# B&R Automation Studio project TD52 (part 97)

#### EG_ScavCyclic.st
```iecst
(*******************************************************************************
EG_Scav			exhaust gas scavenging + N2 scavenging

This code is confidential and proprietary to the INNIO Company.
It may not be used in any form, or reproduced in any manner,
without the express written permission of the INNIO Company.
Copyright, INNIO Company, 2022

Customized modifications: -
------------------------

History:
-------
V06		24.03.2000	PA			erstellt
V11		04.07.2000	Pa			Stoerungsaufbereitung von p10 verschoben
V160	13.12.2001	LH			Ansteuerung Spuelventilator auch mit Gasventile offen
V170	04.02.2002	LH			Moeglichkeit Spuelung manuell zu starten
V190	10.05.2004	LH			Anpassung fuer CODINOX
 								Fehler bei manueller Spuelung ausgebessert
V212	06.06.2006	LH			angepasst an ESY-NEU
V230	12.12.2007	TW			Spuelzeit ist nun Parameter (ssTW_T_SPUEL)
	 	30.01.2008	LH			Untergrenze für Spülzeit ist 47sec
V3.20.0	04.11.2010	lettenb.	purgecycle added, task spuelung renamed to spuelung_6
		14.01.2011 				sel_EGScav_if_AuxV_ok added, release exhaust gas scavenging depending on auxiliaries voltage

V1.70.1	20.03.2003	ThJ			Erweiterung auf N2-Spuelung
V1.70.2	04.05.2004	ThJ			Erweiterung N2-Spuelung von Baureihe 6 auf alle Baureihen
V1.70.3	10.11.2004	ThJ			steps 5 + 8: M_SPUELV hinzu fuer BR234
V1.70.4	15.05.2006	ThJ			Vorbelegung Option "two N2 valves" mit FALSE.
       		              		xx_T71 --> xx_TOF71, xx_T_SPUEL --> xx_TON_SPUEL.
V1.70.5	28.07.2006	ThJ			TwoN2Valves --> global, ANF_SPLV_MAN added,
       		              		N2 gas valves output, N2 valves position faulure modified.
V1.70.6	22.11.2007	ThJ			timer for reset SP_EIN / LUE100
                        		T1_SCAV_RUN: timer 80 --> 75 sec
                        		SCAV_RUN_STOE with filter BWS_A
                        		reset SCAV_RUN at BWS_H by STOP
V1.70.7 03.12.2008	lettenb. 	sel_N2, sel_TwoN2Valves added
V3.40.0	19.12.2012  lettenb.	T1_SCAV_RUN: SCAV_RUN --> STARTER_SC, PT: 75s --> 5s
.								(ueberwachung nun nicht mehr abhaengig von vorschmierzeit/motortemp...., test: SACC, leitner christian)
V3.90.0	25.10.2012	lettenb.	xTON_AuxDemDelayed, Para.bEGScav_Active added
V3.99.0	17.04.2012	lettenb.	EG scav.with all time running fan
		14.05.2013				EG scav.activation for BR6,9 added
		23.10.2013				624: delayed auxiliaries demand with EG scavenging
		28.10.2013				changes from V3.40.1 included, saver case (open flap and fan not demanded) solved
								reset manual scavenging from engine stop button changed > scav.stop button
								N2 scavenging and exhaust gas scavenging merged
		16.01.2014	lettenb.	V3.50 exh.gas scavenging after engine stop with gas train test added
		26.02.2014				tAuxV_Eng_ok.Di added, bugfix
V4.00.0	22.05.2014	lettenb.	T1_STSPKL: scav.valve monitoring open/closed status added, bugfix
V4.00.1 14.07.2014				NoScavFlap, NoScavFan: default = FALSE for EG scav.
		06.08.2014				reset VIS2MM.bN2ScavStart/Stop buttons added
		12.09.2014				SPUEL_ST: AND NOT OUT_EX.bScavFinished added(purge cycle: lock scav.during eng.oper.with eng.dem. off/on)
V4.00.2 30.10.2014	lettenb.	SPUEL_ST: OUT_EX.bScavFinished -> M_DREHZ (purge cycle: lock scav.during eng.oper.)
V4.00.3	20.03.2015	lettenb.	ScavValve opens after bScavFanOp=TRUE, ScavFanCoOn if ScavValve=open or not closed,
								3366 during purge -> close ScavValve(safety case:PW-ER-2015-0062-001)
		14.04.2015				corr.from test EG_Scav with purgecycle and/or purge before start(panian,glantschnig)
		30.04.2015 				OUT_EX.tScavFanCoOn.Do:	IN_EX.tPB2MM.bSys_Run added to avoid bMsg1277 at cold restart
V4.03.0	18.09.2015				IN_EX.bRelEngTurn_OilSkid added for 920
		23.12.2015	lettenb.	OUT_EX.tScavFanCoOn.Do Para.bSel_N2 added, break running scavenging cycle in case of mains break down added,
								to avoid bMsg3366 after mains failure(restart ability)
        02.05.2016              xR_TRIG_M_AGFD: AND NOT M_DREHZ added, to avoid engine shutdown with demand off/on during running engine
V4.04.0 19.09.2016  lettenb.	T1_SCAV_RUN: SCAV_RUN --> STARTER_SC, PT: 75s --> 5s, bugfix, transfer xt4
                                bT1_STN2V: VIS2MM.bEGScavStop -> StopM, bugfix
		14.03.2017	lettenb.	bN2_GASV: OR (NoScavFan AND NoScavFlap) added for BR234(sascha tonauer: U891)
V4.05.0 29.05.2017  lettenb.	fast start preparation: short EG  scavenging(50s) / init EG scavenging if not finished
		12.07.2017  Messner		rT_bScavValve plausibility check added
V4.05.1	16.03.2018	lettenb.	short scavenging only for 920 and only in MAN/AUT, bugfix
		30.07.2018	lettenb.	auto scavenging preparation for faststart
V4.06.0	04.07.2018	Perktold	don't start EGScav for fast start prep. if W3417 is present
V4.07.0 03.12.2018	lettenb.	option NoScavFan completed(SAFER Case ID: PWR-ER-2018-0159), bugfix for option N2 scav.without scav.fan
		13.05.2019	lettenb.	short scavenging only for 920FS for first start sequence, bugfix(request burkhardt wolfg.)
V4.10.0	14.12.2020	lettenb.	TON,TOF reset added to avoid time overrun, cleanup
V4.11.0	14.02.2022	lettenb.	in case of Eng_Dem_EPS wait until running scavenging cycle is finished to avoid engine start with open scavenging flap, bugfix
V4.12.0	14.12.2022	lettenb.	SPUEL_ST: start scavenging when engine is ready4autostart, to avoid scav. at engine demand, #875
								xR_TRIG_M_AGFD: with N2 always scav.before start, #811
								xTON_AB_SPUELV.PT:= T#13s -> 0s (removed in alignment with system owner/burkhart, flap closing is monitored with temp.sensor)
								short scavenging time for FS preparation disabled(not allowed for standard!/TUEV germany)
								calculation of scavenging rest time prepared for HMI display for future(cleanup and learnings from saarbruecken AA46/wasserer)
V4.13.0	05.12.2023	Bacci		Added ventilation demand and release before starting the exhaust scavenging. Reset scavenging procedure when alarm 2295 occurs
V4.14.0	25.11.2024	Bacci		T6 Start procedure with purge start (2024-219): scavenging fan removal

Instructions for use:
--------------------
scavenging fan is always demanded with running engine for cooling of the scav.flap

scavenging functions without N2:
- EG scavenging after  every engine stop
- EG scavenging before every engine start interval if selected
- EG scavenging manual initiated by button
- no EG scavenging after engine stop with emergency stop OR firealarm

scavenging functions with N2:
- EG scavenging before every engine start interval
- EG scavenging manual initiated by button
- N2 scavenging after engine stop
- N2 scavenging after engine startup failure
- N2 scavenging with stopped engine manual initiated by button

observe options: NoScavFlap, NoScavFan, NoPrelube (for engine type 2,3,4)

double ignition: Logical\Ignition\2xzuend\2xzuendCyclic.st
add "AND NOT T_N2_GASV" to avoid ignition failure during stand still N2 scavenging
		(* Ignition 1 error
		xTONIgn1FaultDelay(IN:= NOT IN_IG.bIgn_Dem AND IN_IG.tIgn_Run_Hal.Di, PT:=T#4s);
		ZEST_1 :=  (xTONIgn1FaultDelay.Q AND NOT T_N2_GASV)
				OR (IN_IG.bGV_On AND NOT IN_IG.bMsg1026 AND IN_IG.bIgn_Dem AND NOT IN_IG.tIgn_Run_Hal.Di);

		(* Ignition 2 error
		xTONIgn2FaultDelay(IN:= NOT IN_IG.bIgn_Dem AND IN_IG.tIgn2_Run_Hal.Di, PT:=T#4s);
		ZEST_2 :=  (xTONIgn2FaultDelay.Q AND NOT T_N2_GASV)
				OR (IN_IG.bGV_On AND NOT IN_IG.bMsg1026 AND IN_IG.bIgn_Dem AND NOT IN_IG.tIgn2_Run_Hal.Di);

		(* flag for deactivating gas pressure monitoring
		xTOF_T_N2_GASV(IN:= OUT_EX.tN2_ScavGV_CoOpen.Do, PT:= T#5s);
		T_N2_GASV := xTOF_T_N2_GASV.Q;

Outstandings:
------------
*******************************************************************************)
PROGRAM _CYCLIC

	(* Engine speed is below 50 rpm *)
	IF (IN_EX.rN_EngAct < 50.0) THEN	StopM := TRUE;
	ELSE								StopM := FALSE;
	END_IF;

	(* prelube oil pressure 1 *)
	xGR_MAXR_VSD1(In:= IN_EX.tPr_EngLubOil.Ai, Gw:= Para.rPr_Prel1EOP_LimHi, Hy:= Para.rPr_Prel1EOP_HyHi);
	xTON_VSD1(IN:= xGR_MAXR_VSD1.Q AND IN_EX.tPB2MM.bParaSetupOk, PT:= T#2s);
	AN_VSD1 := xTON_VSD1.Q;

	(* speed limit *)
	xGR_MAXR_D1400(In:= IN_EX.rN_EngAct, Gw:= (Para.rN_EngNom - 100.0), Hy:= 10.0);
	M_D1400	:= xGR_MAXR_D1400.Q;

	(* Monitoring engine start speed  *)
	xGR_MAXR_MonEngStaSpeed(In:= IN_EX.rN_EngAct, Gw:= Para.rN_EngStartMon_LimHi, Hy:= Para.rN_EngStartMon_HyHi);
	AN_STRDRE :=  IN_EX.tPB2MM.bParaSetupOk AND xGR_MAXR_MonEngStaSpeed.Q;

	(* engine start speed *)
	xGR_MAXR_EngStaSpeed(In:= IN_EX.rN_EngAct, Gw:= Para.rN_EngStart_LimHi, Hy:= Para.rN_EngStart_HyHi);
	xTOF_MDREHZ(IN:= IN_EX.tPB2MM.bParaSetupOk AND xGR_MAXR_EngStaSpeed.Q, PT:= T#10s);
	M_DREHZ    := xTOF_MDREHZ.Q;

	(*-----------------------------------------------------------------------------------------------------*)
	(*-----------------------------------------------------------------------------------------------------*)
	(* manual demand exhaust gas scavenging *)
	VIS2MM.bEGScavStart;	VIS2MM.bEGScavStop;

	(* manual demand N2 gas scavenging *)
	VIS2MM.bN2ScavStart;	VIS2MM.bN2ScavStop;

	(* scavenging valve feedback signals *)
	bScavVaIsOpened :=	IN_EX.tScavVaOpened.Di AND NOT IN_EX.tScavVaClosed.Di; (* scav.valve = opened *)
	bScavVaIsClosed :=	IN_EX.tScavVaClosed.Di AND NOT IN_EX.tScavVaOpened.Di; (* scav.valve = closed *)

	(* scavenging fan operating *)(**)
	bScavFanOp :=	(NOT xEngType.Type9 AND(IN_EX.tScavFanOp.Di OR NoScavFan))
				OR	(    xEngType.Type9 AND(IN_EX.tScavFanFC_Rdy.Di AND NOT IN_EX.tScavFanFC_P_Lo.Di));

	(*-----------------------------------------------------------------------------------------------------*)
	IF Para.bEGScav_Active OR Para.bSel_N2 OR xEngType.Type9  THEN	(* exhaust gas scavenging with N2 *)

		OUT_EX.bRel_ScavN2 :=	Para.bSel_N2
						AND(    IN_EX.bGT2_Select OR NOT Para.bN2_NoScavGas1)
						AND(NOT IN_EX.bGT2_Select OR NOT Para.bN2_NoScavGas2);

		(* option: no scavenging fan/flap *)
		NoScavFlap := FALSE;	//xEngType.Type2 OR xEngType.Type3 OR xEngType.Type4;
		NoScavFan  := FALSE;	//xEngType.Type2 OR xEngType.Type3 OR xEngType.Type4;

		(* option: no prelubrication *)
		NoPrelube  := xEngType.Type3 AND NOT Para.bEngTyp3_Prelub_Active;

		(* scavenging initiated by startup failure/error *)
		SCAV_RUN_STOE := IN_EX.bMsg1023 AND bOMSS_Aut;

		FG_SCAV_RUN :=	OUT_EX.bRel_ScavN2
				AND NOT M_DREHZ
				AND NOT IN_EX.bMsg1031
				AND NOT IN_EX.bMsg1054
				AND NOT IN_EX.bMsg1060
			    AND NOT IN_EX.bMsg1108
				AND NOT IN_EX.bMsg1084
				AND NOT IN_EX.bMsg1056;

		FG_SCAV_RUN_2 :=	FG_SCAV_RUN
					AND 	StopM
					AND	  ((bOMSS_Scav AND VIS2MM.bN2ScavStart) OR (SCAV_RUN_STOE AND NOT M_SCAV_RUN));

		xTON_SCR_OFF1(IN:= OUT_EX.bN2_ScavCoStarterOn, PT:= T#20s);

		IF     (NOT FG_SCAV_RUN
			OR (    bOMSS_Scav AND     VIS2MM.bN2ScavStop)
			OR (NOT bOMSS_Scav AND NOT bOMSS_MAT)
			OR (    bOMSS_Man  AND     VIS2MM.bN2ScavStop)
			OR (    bOMSS_Aut  AND NOT SCAV_RUN_STOE)
			OR	    T2_SCAV_RUN
			OR	    xTON_SCR_OFF1.Q) THEN	SCAV_RUN := FALSE;
		ELSIF FG_SCAV_RUN_2 THEN			SCAV_RUN := TRUE;
			IF SCAV_RUN_STOE THEN			M_SCAV_RUN := TRUE;
			END_IF;
		END_IF;

		IF NOT SCAV_RUN_STOE THEN
			M_SCAV_RUN := FALSE;
		END_IF;

		(*-------------------------------------------------------------------*)
		(* lockout scavenging after engine stop in case of: *)
		bNoScavAftEngStop := 	IN_EX.bMsg1031
							OR	IN_EX.bMsg1054;

		(* short scavenging time for FS preparation *)
		IF IN_EX.tEng_Run.Do       THEN bFS_ScavTime := FALSE; (* not allowed for standard! *)
//		IF IN_EX.tEng_Run.Do       THEN bFS_ScavTime := TRUE;  (* enable only with special release, incl. risk analysis approval *)
		ELSIF IN_EX.bGV_On         THEN bFS_ScavTime := FALSE;
		END_IF;

		(* set/reset purge credit bit = bScavFinished *)
		xF_TRIG_M_GASV(CLK:= IN_EX.bGV_On);
		xR_TRIG_M_AGFD(CLK:= IN_EX.bEng_Dem AND NOT M_DREHZ AND (Para.bScavBeStart_Active OR Para.bSel_N2));

		IF 	  IN_EX.bEng_Dem_EPS AND(NOT Para.bEGScav_ifAuxV_ok OR NOT IN_EX.tAuxV_Eng_ok.Di) AND (StepCnt = 0)
														THEN OUT_EX.bScavFinished := 1; (*needed for emerg.power supply after plc-restart ! *)
		ELSIF bNoScavAftEngStop 						THEN OUT_EX.bScavFinished := 0; (* scavening after engine stop not released *)
															 bFS_ScavTime := FALSE;
		ELSIF xF_TRIG_M_GASV.Q							THEN OUT_EX.bScavFinished := 0; (* gas valves closed *)
		ELSIF xR_TRIG_M_AGFD.Q							THEN OUT_EX.bScavFinished := 0; (* scavenging before start *)
		ELSIF MM2VIS.bMsg3417   AND NOT IN_EX.bEng_Dem	THEN OUT_EX.bScavFinished := 0; (* pre chamber diff.press.high during engine stop (exh.gas scav.required before next start)*)
															 bFS_ScavTime := FALSE;
		ELSIF EDGEPOS(IN_EX.bMsg1084)					THEN OUT_EX.bScavFinished := 0;	(* signal failure prechamber gas pressure *)
															 bFS_ScavTime := FALSE;
		ELSIF EDGEPOS(IN_EX.bMsg1056)					THEN OUT_EX.bScavFinished := 0; (* safety loop engine *)
															 bFS_ScavTime := FALSE;
		ELSIF EDGEPOS(IN_EX.bMsg1027)					THEN OUT_EX.bScavFinished := 0; (* failure gas train 1 -(line 1)*)
															 bFS_ScavTime := FALSE;
		ELSIF EDGEPOS(IN_EX.bMsg3361)					THEN OUT_EX.bScavFinished := 0; (* failure gas train 1 - line 4 *)
															 bFS_ScavTime := FALSE;
		ELSIF EDGEPOS(IN_EX.bMsg3360)					THEN OUT_EX.bScavFinished := 0; (* failure gas train 1 - line 3 *)
															 bFS_ScavTime := FALSE;
		ELSIF EDGEPOS(IN_EX.bMsg3359)					THEN OUT_EX.bScavFinished := 0; (* failure gas train 1 - line 2 *)
															 bFS_ScavTime := FALSE;
		ELSIF EDGEPOS(IN_EX.bMsg1029)					THEN OUT_EX.bScavFinished := 0; (* failure gas train 2 *)
															 bFS_ScavTime := FALSE;
		ELSIF MM2VIS.bMsg3366							THEN OUT_EX.bScavFinished := 0; (* exhaust gas scavening fan failure BR2346 *)
															 bFS_ScavTime := FALSE;
		ELSIF MM2VIS.bMsg1165							THEN OUT_EX.bScavFinished := 0; (* exhaust gas scavening fan failure BR9 *)
															 bFS_ScavTime := FALSE;
		ELSIF MM2VIS.bMsg1092							THEN OUT_EX.bScavFinished := 0; (* exhaust gas scavening valve failure *)
															 bFS_ScavTime := FALSE;
		ELSIF EDGEPOS(IN_EX.tPB2MM.bSys_Run)			THEN OUT_EX.bScavFinished := 0; (* plc restart *)
															 bFS_ScavTime := FALSE;
		END_IF;

		(*-------------------------------------------------------------------*)
		IF bOMSS_MAT AND NOT M_DREHZ AND (IN_EX.tEGScavStart_Ext.Di OR VIS2MM.bEGScavStart) THEN
			MAN_SPUEL := TRUE;
		END_IF;
		xTOF_MAN_SPUEL(IN:= MAN_SPUEL, PT:= T#2s);

		xTON_AutStartPrep(IN:= bOMSS_Aut AND NOT bGnlTrip AND NOT IN_EX.bEng_Dem AND NOT Para.bScavBeStart_Active AND NOT Para.bSel_N2, PT:= T#60s); (* do scavenging for auto start preparation *)

		(* scavenging start *)
 		SPUEL_ST :=	   (bOMSS_MAT
				AND NOT	MM2VIS.bMsg1165
				AND NOT MM2VIS.bMsg3417
				AND    (IN_EX.bEng_Dem
					OR  xTON_AutStartPrep.Q
					OR (IN_EX.bFS_Act AND bOMSS_Aut))
				AND NOT OUT_EX.bScavFinished
				AND    (IN_EX.bPurgeER_Rdy OR NOT Para.bPurgecycle_Active))
			OR  xTOF_MAN_SPUEL.Q;

		(* scavenging before engine start *)
		SCAV_BEF :=		SPUEL_ST
				AND NOT M_DREHZ
				AND(NOT IN_EX.bEng_Dem_EPS OR (Para.bEGScav_ifAuxV_ok AND IN_EX.tAuxV_Eng_ok.Di)); 	(* no scav.in case of demand emergency supply *)

		(* scavenging after engine stop *)
		SCAV_AFT := FALSE;
		IF (T1_StopM AND FG_SCAV_AFT AND NOT SCAV_RUN) THEN
			SCAV_AFT    := T1_StopM AND FG_SCAV_AFT AND NOT SCAV_RUN AND NOT bNoScavAftEngStop;
			FG_SCAV_AFT := FALSE;
		ELSIF (NOT StopM AND (M_DREHZ OR SCAV_RUN) AND (OUT_EX.bRel_ScavN2 OR TRUE)) THEN
			FG_SCAV_AFT := TRUE;
		END_IF;

		(*-------------------------------------------------------------*)
		IF EDGEPOS(SCAV_BEF OR SCAV_AFT) AND NOT bNoScavAftEngStop THEN
			OUT_EX.bScavFinished := FALSE;				(* = engine start release = purge credit bit *)
			StepCnt 		:= 10;
		ELSIF NOT IN_EX.tAuxV_Eng_ok.Di THEN			(* break running scavenging cycle in case of mains break down during scavenging*)
			StepCnt 		:= 0;
		ELSIF IN_EX.bMsg1031 OR IN_EX.bMsg1054 OR MM2VIS.bMsg1092 OR MM2VIS.bMsg3366 OR IN_EX.bMsg2295 THEN	(* break running scavenging cycle *)
			StepCnt 		:= 0;
		ELSIF MAN_SPUEL AND VIS2MM.bEGScavStop THEN		(* break running man.scavenging cycle *)
			StepCnt 		:= 0;
		END_IF;

		(*----------------------------------------------------------------*)
		IF StepCnt = 0 THEN
			M_SPUELV			:= FALSE;
			OUT_EX.bDemScavVa	:= FALSE;
			MAN_SPUEL			:= FALSE;
			xTON_T_SPUEL(IN:= FALSE, PT:= T#0s); (* reset timer out of stepper loop *)
			xTON_AB_SPUELV(IN:= FALSE, PT:= T#0s); (* reset timer out of stepper loop *)
			xTON_P_SPUEL(IN:= FALSE, PT:= T#0s); (* reset timer out of stepper loop *)
		END_IF;

		(*----------------------------------------------------------------*)
		(* Step 1: Open scavenging valve *)
		IF StepCnt = 10 THEN
			M_SPUELV 			:= TRUE;(**)

			IF bScavFanOp OR NoScavFan THEN
				OUT_EX.bDemScavVa := TRUE;
				StepCnt := StepCnt + 10;
			END_IF;
		END_IF;

		(*----------------------------------------------------------------*)
		(* Step 2: Scavenging period *)
		IF StepCnt = 20 THEN

			IF (IN_EX.bFS_Act AND xEngType.Type9 AND bFS_ScavTime) THEN
					xTON_T_SPUEL.PT:= T#50s;			(* fast start scavenging time *)
					xTON_T_SPUEL(IN:=	OUT_EX.bDemScavVa
									AND	M_SPUELV);
			ELSE	xTON_T_SPUEL.PT:= Para.tiEGScavMin; (* standard   scavenging time *)
					xTON_T_SPUEL(IN:=	OUT_EX.bDemScavVa
									AND(bScavVaIsOpened OR NoScavFlap)
									AND	M_SPUELV);
			END_IF;
			IF xTON_T_SPUEL.Q THEN
				OUT_EX.bDemScavVa := FALSE;
				StepCnt := StepCnt + 10;
			END_IF;
		END_IF;

		(*----------------------------------------------------------------*)
		(* Step 3: waiting period until scavenging valve is completly closed*)
		(*         scavenging fan off *)
		IF StepCnt = 30 THEN
			IF (IN_EX.bFS_Act AND xEngType.Type9 AND bFS_ScavTime) THEN
					xTON_AB_SPUELV.PT:= T#0s;  (* fast start scavenging *)
			ELSE	xTON_AB_SPUELV.PT:= T#0s;  (* standard   scavenging *)
			END_IF;
			xTON_AB_SPUELV(IN:= NOT OUT_EX.bDemScavVa AND (    bScavVaIsClosed OR NoScavFlap));
			xTON_CloScavVa(IN:= NOT OUT_EX.bDemScavVa AND (NOT bScavVaIsClosed OR NoScavFlap), PT:=T#15s); (* scav.flap estimated closing time for rest time calculation *)
			IF xTON_AB_SPUELV.Q THEN
				M_SPUELV := FALSE;
				StepCnt := StepCnt + 10;
			END_IF;
		END_IF;

		(*----------------------------------------------------------------*)
		(* Step 4: exhaust gas scavenging completed, release engine startup *)
		IF StepCnt = 40 THEN
			IF (IN_EX.bFS_Act AND xEngType.Type9 AND bFS_ScavTime) THEN
					xTON_P_SPUEL.PT:= T#0s; (* fast start scavenging *)
			ELSE	xTON_P_SPUEL.PT:= T#2s; (* standard   scavenging *)
			END_IF;
			xTON_P_SPUEL(IN:= NOT OUT_EX.bDemScavVa AND(bScavVaIsClosed OR NoScavFlap));

			IF xTON_P_SPUEL.Q AND (xTON_SCAV_OFF.Q OR NOT Para.bSel_N2) THEN (* +60s room ventilation at 100% when N2 scavenging *)
				OUT_EX.bScavFinished := TRUE;(* no scav.fan+valve failure! -> scav.is done*)(**)
				StepCnt := 0;
			END_IF;
		END_IF;

		(* calculation of scavenging rest time *)
		MM2VIS.bScavRun := xTON_T_SPUEL.IN OR OUT_EX.bDemScavVa OR (xTON_SCAV_OFF.IN AND Para.bSel_N2);
		IF MM2VIS.bScavRun THEN MM2VIS.tiScavRestTime := ((xTON_T_SPUEL.PT   - xTON_T_SPUEL.ET  )/1000)
								                       + ((xTON_AB_SPUELV.PT - xTON_AB_SPUELV.ET)/1000)
													   +(((xTON_CloScavVa.PT - xTON_CloScavVa.ET)/1000) * BOOL_TO_INT(NOT bScavVaIsClosed))
													   +(((xTON_SCAV_OFF.PT  - xTON_SCAV_OFF.ET )/1000) * BOOL_TO_INT(Para.bSel_N2));
		ELSE
			MM2VIS.tiScavRestTime := 0;
		END_IF

		(*----------------------------------------------------------------*)
		(*----------------------------------------------------------------*)
		(* command open/close scavenging valve  *)
		bScavVaCoOpen  := NOT MM2VIS.bMsg1092 AND     OUT_EX.bDemScavVa AND NOT bScavVaCoClose;
		bScavVaCoClose := NOT MM2VIS.bMsg1092 AND NOT OUT_EX.bDemScavVa AND NOT bScavVaCoOpen;

		xTON_SPKAUF(IN:= bScavVaCoOpen,  PT:= T#0.5s);
		xTON_SPKZU (IN:= bScavVaCoClose, PT:= T#0.5s);

		OUT_EX.tScavVaCoOpen.Do  := xTON_SPKAUF.Q;
		OUT_EX.tScavVaCoClose.Do := xTON_SPKZU.Q;

		(* scavenging valve failure*)
		xTON_T1_STSPKL(IN:= IN_EX.tPB2MM.bSys_Run
					AND     IN_EX.tPB2MM.bParaSetupOk
					AND	  ((OUT_EX.tScavVaCoOpen.Do  AND NOT NoScavFlap AND NOT bScavVaIsOpened)
						OR (OUT_EX.tScavVaCoOpen.Do  AND NOT NoScavFlap AND     bScavVaIsClosed)
						OR (OUT_EX.tScavVaCoClose.Do AND NOT NoScavFlap AND NOT bScavVaIsClosed)
						OR (OUT_EX.tScavVaCoClose.Do AND NOT NoScavFlap AND     bScavVaIsOpened)), PT:= T#35s);
		T1_STSPKL := xTON_T1_STSPKL.Q; (* valve runtime monitoring *)

		xTON_T2_STSPKL(IN:= NOT IN_EX.tScavVaFailure.Di AND NOT NoScavFlap, PT:= T#2s);
		T2_STSPKL := xTON_T2_STSPKL.Q; (* temperature monitoring *)

		(* scavenging fan at engine operation *)
		IF    IN_EX.bGV_On  OR SCAV_RUN THEN	BETR_SPUELV := TRUE;
		ELSIF T2_StopM AND NOT SCAV_RUN THEN	BETR_SPUELV := FALSE;
		END_IF;

		OUT_EX.bInLouDemEX :=			IN_EX.tPB2MM.bSys_Run (* inlet louver demand *)
								AND	NOT	NoScavFan
								AND		(M_SPUELV OR(BETR_SPUELV AND Para.bSel_N2) OR(NOT NoScavFlap AND(IN_EX.tScavVaOpened.Di OR NOT IN_EX.tScavVaClosed.Di)));

		(* DO scavenging fan on *)
		OUT_EX.tScavFanCoOn.Do :=	(OUT_EX.bInLouDemEX AND IN_EX.bInLouRelVE) OR
									(IN_EX.tPB2MM.bSys_Run AND NOT NoScavFan AND IN_EX.bGV_On) OR
									(IN_EX.tPB2MM.bSys_Run AND NOT NoScavFan AND (NOT NoScavFlap AND(IN_EX.tScavVaOpened.Di OR NOT IN_EX.tScavVaClosed.Di)));

		(* Signal lamp scavenging *)
		(* Engine room ventilation at 100% *)
		xTON_SCAV_OFF(IN:= T2_StopM AND NOT SCAV_RUN, PT:= T#60s);

		IF (SCAV_RUN OR M_SPUELV OR (NOT StopM AND M_DREHZ AND NOT IN_EX.bGV_On)) THEN
			OUT_EX.tN2_ScavSigLampOn.Do := TRUE;
			OUT_EX.bInAirER_FanSet100   := TRUE;
		ELSIF (NOT M_SPUELV AND xTON_SCAV_OFF.Q) THEN
			OUT_EX.tN2_ScavSigLampOn.Do := FALSE;
			OUT_EX.bInAirER_FanSet100   := FALSE;
		END_IF;

		(* N2 gas valves for scavenging *)
		(* time delay for waiting during closing time of the gas valves *)
		bZM_N2_GASV :=	   (IN_EX.tScavVaClosed.Di OR NoScavFlap)
					AND	NOT OUT_EX.bPr_N2_LoTon
					AND 	OUT_EX.bRel_ScavN2
					AND	   (IN_EX.tEG_ByVaOpened.Di OR IN_EX.tEG_BoVaOpened.Di);

		(* N2 gas valves not for BR2,3,4 if nominal speed was reached (V1.70.2)*)
		xTON_DREHZ_N2(IN:= M_DREHZ AND M_D1400, PT:= T#10s);
		IF xTON_DREHZ_N2.Q THEN M_DREHZ_N2 := TRUE;	// xSR_FA_M_DREHZ_N2 --> M_DREHZ_N2
		ELSIF NOT M_DREHZ  THEN M_DREHZ_N2 := FALSE;
		END_IF;

		bN2_GASV := 	bZM_N2_GASV
				AND NOT StopM
				AND NOT IN_EX.bGV_On
				AND    (SCAV_RUN OR (M_DREHZ  AND (NOT M_DREHZ_N2
                                                   OR  xEngType.Type6
                                                   OR  xEngType.Type9
                                                   OR (NoScavFan AND NoScavFlap))));//BR234

		xTON_N2_GASV(IN:= bN2_GASV, PT:= T#1s);

		(* switch N2 Gas Valve with reset as priority *)
		IF     (StopM
			OR  IN_EX.bGV_On
			OR (NOT IN_EX.tScavVaClosed.Di AND NOT NoScavFlap)
			OR  OUT_EX.bPr_N2_LoTon
			OR  NOT OUT_EX.bRel_ScavN2
			OR (NOT IN_EX.tEG_ByVaOpened.Di AND NOT IN_EX.tEG_BoVaOpened.Di)) THEN
		    OUT_EX.tN2_ScavGV_CoOpen.Do := FALSE;
		ELSIF xTON_N2_GASV.Q THEN
			OUT_EX.tN2_ScavGV_CoOpen.Do := TRUE;
		END_IF;

		(* flag for deactivating gas pressure monitoring *)
		xTOF_T_N2_GASV(IN:= OUT_EX.tN2_ScavGV_CoOpen.Do, PT:= T#5s);
		T_N2_GASV := xTOF_T_N2_GASV.Q;

		(* scavenging run of the engine (prelub. + starter) *)
		IF NOT SCAV_RUN THEN
			OUT_EX.bN2_ScavCoStarterOn := FALSE;
			IF T1_StopM THEN
				OUT_EX.bN2_ScavCoPrelubeOn := FALSE;
			END_IF;
			xTON_START_SC(IN:= FALSE, PT:= T#0s);
		ELSE
			OUT_EX.bN2_ScavCoPrelubeOn := TRUE;
			IF xEngType.Type9 THEN 	xTON_START_SC(IN:=  AN_VSD1 AND IN_EX.bRelEngTurn_OilSkid, PT:= T#60s);
			ELSE					xTON_START_SC(IN:=  AN_VSD1 OR NoPrelube,                  PT:= T#60s);
			END_IF;

			IF xTON_START_SC.Q THEN
				OUT_EX.bN2_ScavCoStarterOn := TRUE;
			END_IF;
		END_IF;

		(* monitoring --------------------------------------------------*)
		(* N2 valves position failure *)
		IF Para.bSel_TwoN2Valves THEN
			bN2_GV_AnyClosed :=     IN_EX.tN2_GV1_Closed.Di OR      IN_EX.tN2_GV2_Closed.Di;
			bN2_GV_AnyOpened := NOT IN_EX.tN2_GV1_Closed.Di OR  NOT IN_EX.tN2_GV2_Closed.Di;
		ELSE
			bN2_GV_AnyClosed :=     IN_EX.tN2_GV1_Closed.Di;
			bN2_GV_AnyOpened := NOT IN_EX.tN2_GV1_Closed.Di;
		END_IF;

		bT1_STN2V	 := 	OUT_EX.bRel_ScavN2
					AND NOT StopM
					AND 	M_DREHZ
					AND NOT IN_EX.bGV_On
					AND(NOT M_DREHZ_N2 OR xEngType.Type6 OR xEngType.Type9);

		xTON_T1_STN2V(IN:= (	OUT_EX.tN2_ScavGV_CoOpen.Do AND bN2_GV_AnyClosed)
						OR (	bT1_STN2V					AND bN2_GV_AnyClosed)
						OR (NOT OUT_EX.tN2_ScavGV_CoOpen.Do AND bN2_GV_AnyOpened), PT:= T#5s);

		xTON_T2_STN2V(IN:=	IN_EX.bGV_On AND bN2_GV_AnyOpened, PT:= T#500ms);

		T1_STN2V := xTON_T1_STN2V.Q OR xTON_T2_STN2V.Q OR (NOT IN_EX.tEG_ByVaOpened.Di AND NOT IN_EX.tEG_BoVaOpened.Di);

		(* monitoring N2 gas valves position *)
		xTON_T1_SCAV_RUN(IN:= OUT_EX.bN2_ScavCoStarterOn AND bN2_GV_AnyClosed, PT:= T#5s);
		T1_SCAV_RUN := xTON_T1_SCAV_RUN.Q;

		(* monitoring scavenging time *)
		xTON_T2_SCAV_RUN(IN:= SCAV_RUN, PT:= T#120s);
		T2_SCAV_RUN := xTON_T2_SCAV_RUN.Q;

		(* N2 gas pressure minimum *)
		xTON_GDMI_N2(IN:= NOT IN_EX.tPr_N2_Lo.Di, PT:= T#5s);
		OUT_EX.bPr_N2_LoTon := xTON_GDMI_N2.Q;

		(* timer for engine standstill time from 50 rpm -> 0 rpm *)
		xTON_T1_StopM(IN:= StopM, PT:= T#4s);
		T1_StopM := xTON_T1_StopM.Q;

		(* Timer for overlapping with the start of "scavenging after engine stop" *)
		xTON_T2_StopM(IN:= StopM, PT:= Para.tiEGScavMin);
		T2_StopM := xTON_T2_StopM.Q;

	(*-----------------------------------------------------------------------------------------------------*)
		(* Scavenging fan set-point *)
		IF (OUT_EX.tScavFanCoOn.Do AND IN_EX.tScavVaClosed.Di) THEN
			OUT_EX.tScavFan_Sp.Ao := 0.0;
		ELSE
			OUT_EX.tScavFan_Sp.Ao := 1.0;
		END_IF;

	(*-----------------------------------------------------------------------------------------------------*)
	ELSE (* no exhaust gas scavenging *)
		xTON_SCR_OFF1(IN:= FALSE, PT:= T#0s);
		xTON_T_SPUEL(IN:= FALSE, PT:= T#0s);
		xTON_AB_SPUELV(IN:= FALSE, PT:= T#0s);
		xTON_P_SPUEL(IN:= FALSE, PT:= T#0s);
		xTON_SPKAUF(IN:= FALSE,  PT:= T#0s);
		xTON_SPKZU(IN:= FALSE, PT:= T#0s);
		xTON_T1_STSPKL(IN:= FALSE, PT:= T#0s);
		xTON_T2_STSPKL(IN:= FALSE, PT:= T#0s);
		xTON_SCAV_OFF(IN:= FALSE, PT:= T#0s);
		xTON_DREHZ_N2(IN:= FALSE, PT:= T#0s);
		xTON_N2_GASV(IN:= FALSE, PT:= T#0s);
		xTON_START_SC(IN:= FALSE, PT:= T#0s);
		xTON_T1_STN2V(IN:= FALSE, PT:= T#0s);
		xTON_T2_STN2V(IN:= FALSE, PT:= T#0s);
		xTON_T1_SCAV_RUN(IN:= FALSE, PT:= T#0s);
		xTON_T2_SCAV_RUN(IN:= FALSE, PT:= T#0s);
		xTON_GDMI_N2(IN:= FALSE, PT:= T#0s);
		xTON_T1_StopM(IN:= FALSE, PT:= T#0s);
		xTON_T2_StopM(IN:= FALSE, PT:= T#0s);

		xTOF_MAN_SPUEL(IN:= FALSE, PT:= T#0s);
		xTOF_T_N2_GASV(IN:= FALSE, PT:= T#0s);

		OUT_EX.bRel_ScavN2 := FALSE;
		OUT_EX.bScavFinished := TRUE;

	END_IF;

	(*---------------------------------------------------------------------------------------*)
	(* delayed auxiliaries demand with EG scavenging --> MM_OP *)
	IF xEngType.Type9 THEN
		IF Para.tiEGScavMin <= T#60s THEN	xTON_AuxDemDelayed.PT := T#0s;
		ELSE								xTON_AuxDemDelayed.PT := Para.tiEGScavMin - T#60s;
		END_IF;
	ELSIF Para.iEng_Motortype = 624 THEN
		IF Para.tiEGScavMin <= T#120s THEN	xTON_AuxDemDelayed.PT := T#0s;
		ELSE								xTON_AuxDemDelayed.PT := Para.tiEGScavMin - T#120s;
		END_IF;
	ELSE
		IF Para.tiEGScavMin <= T#60s THEN	xTON_AuxDemDelayed.PT := T#0s;
		ELSE								xTON_AuxDemDelayed.PT := Para.tiEGScavMin - T#60s;
		END_IF;
	END_IF;

	xTON_AuxDemDelayed(IN:= IN_EX.bEng_Dem);

	OUT_EX.bEGScav_Rdy := xTON_AuxDemDelayed.Q OR OUT_EX.bScavFinished;

	(********************************************************************************************************************
	Safety-related application software source code (EN 13849-1 / 4.6.3): BEGIN
	*********************************************************************************************************************)
	(* Measuring Signal Plausibility Check - air temperature before exhaust gas scavening valve (Functional Safety) *)

	(* Timer for Engine Run and Engine Stop *)
	xTON_EngRun (IN:= IN_EX.tEng_Run.Do, PT:= T#10m);
	xTON_EGScav	(IN:= bTON_EngRun AND bScavVaIsOpened, PT:= T#25s);

	(* Set and Reset - Engine Run State *)
	IF xTON_EngRun.Q 			THEN bTON_EngRun := TRUE;	END_IF;	(* Engine Running for given time *)
	IF EDGENEG(bScavVaIsOpened) THEN bTON_EngRun := FALSE; 	END_IF;	(* Falling Edge om Scavenging Fan ON *)

	(* Rising Edge on Engine Timer *)
	xR_TRIG_StorePreEGScavValue (CLK:= IN_EX.tPB2MM.bSys_Run AND bTON_EngRun AND OUT_EX.tScavVaCoOpen.Do);
	xR_TRIG_StoreAftEGScavValue (CLK:= IN_EX.tPB2MM.bSys_Run AND xTON_EGScav.Q);

	(* Save Variables on lokal Storage *)
	IF xR_TRIG_StorePreEGScavValue.Q 	THEN rT_bScavValve_PreEGScavValue := IN_EX.tT_bScavValve.Ai;
	END_IF;
	IF xR_TRIG_StoreAftEGScavValue.Q 	THEN rT_bScavValve_AftEGScavValue := IN_EX.tT_bScavValve.Ai;
	END_IF;

	(* Reset Saved Values if Warning Reset*)
	IF bT_bScavValve_PcheckFail AND IN_EX.tAB2EX.bResetWarning THEN
		rT_bScavValve_PreEGScavValue 	:= 0.0;
		rT_bScavValve_AftEGScavValue 	:= 0.0;
	END_IF;

	(* Set Trigger Variable *)
	IF MM2VIS.bMsg2468 THEN															bT_bScavValve_PcheckFail := FALSE;
	ELSIF (rT_bScavValve_PreEGScavValue = 0.0) THEN									bT_bScavValve_PcheckFail := FALSE; 	(* value not valid *)
	ELSIF (rT_bScavValve_AftEGScavValue = 0.0) THEN									bT_bScavValve_PcheckFail := FALSE; 	(* value not valid *)
	ELSE
		IF (rT_bScavValve_PreEGScavValue - rT_bScavValve_AftEGScavValue) < 5 THEN	bT_bScavValve_PcheckFail := TRUE;	(* Air temperature changed less then 5°C *)
		END_IF;

		IF xR_TRIG_StoreAftEGScavValue.Q THEN			(* Reset saved temperatures - Valve closes *)
			rT_bScavValve_PreEGScavValue 	:= 0.0;
			rT_bScavValve_AftEGScavValue 	:= 0.0;
		END_IF;
	END_IF;

	(*---------------------------------------------------------------------------------------*)
	(* reset VIS2MM var. *)
	VIS2MM.bEGScavStart := FALSE;
	VIS2MM.bEGScavStop  := FALSE;
	VIS2MM.bN2ScavStart := FALSE;
	VIS2MM.bN2ScavStop  := FALSE;
	(********************************************************************************************************************
	Safety-related application software source code (EN 13849-1 / 4.6.3): END
	*********************************************************************************************************************)

END_PROGRAM
```

#### EG_Scav.var
```iecst
VAR
	bScavVaCoOpen : BOOL := 0; (*scavenging valve command open*)
	bScavVaCoClose : BOOL := 0; (*scavenging valve command close*)
	bScavVaIsOpened : BOOL := 0; (*scavenging valve is opened*)
	bScavVaIsClosed : BOOL := 0; (*scavenging valve is closed*)
	NoPrelube : BOOL := FALSE;
	SCAV_AFT : BOOL := FALSE;
	FG_SCAV_RUN_2 : BOOL;
	FG_SCAV_RUN : BOOL := FALSE;
	M_SCAV_RUN : BOOL := FALSE;
	SCAV_BEF : BOOL := FALSE;
	T1_StopM : BOOL := FALSE;
	SCAV_RUN_STOE : BOOL := FALSE;
	SCAV_RUN : BOOL := FALSE;
	T_N2_GASV : BOOL;
	BETR_SPUELV : BOOL := FALSE;
	AN_STRDRE : BOOL;
	bZM_N2_GASV : BOOL;
	FG_SCAV_AFT : BOOL := FALSE;
	T2_StopM : BOOL := FALSE;
	xGR_MAXR_EngStaSpeed : GR_MAXR := (0);
	xGR_MAXR_D1400 : GR_MAXR;
	xGR_MAXR_MonEngStaSpeed : GR_MAXR := (0);
	xGR_MAXR_VSD1 : GR_MAXR;
	xTOF_MDREHZ : TOF := (0);
	xTON_P_SPUEL : TON;
	xTON_SCAV_OFF : TON := (0);
	xTON_T1_STSPKL : TON;
	xTON_T2_STSPKL : TON;
	xTON_SCR_OFF1 : TON;
	xTON_SPKAUF : TON := (0);
	xTON_VSD1 : TON;
	xTON_SPKZU : TON := (0);
	xTON_AuxDemDelayed : TON;
	xTOF_MAN_SPUEL : TOF;
	xTON_DREHZ_N2 : TON;
	bN2_GASV : BOOL;
	xTON_N2_GASV : TON;
	xTOF_T_N2_GASV : TOF;
	xTON_START_SC : TON;
	bN2_GV_AnyClosed : BOOL;
	bN2_GV_AnyOpened : BOOL;
	bT1_STN2V : BOOL;
	xTON_T2_STN2V : TON;
	xTON_T1_STN2V : TON;
	xTON_T1_SCAV_RUN : TON;
	xTON_T2_SCAV_RUN : TON;
	xTON_GDMI_N2 : TON;
	xTON_T1_StopM : TON;
	xTON_T2_StopM : TON;
	M_DREHZ_N2 : BOOL;
	xF_TRIG_M_GASV : F_TRIG;
	xR_TRIG_M_AGFD : R_TRIG;
	StepCnt : INT;
	bNoScavAftEngStop : BOOL;
	xTON_T_SPUEL : TON;
	xTON_AB_SPUELV : TON;
	SPUEL_ST : BOOL := 0; (*Scavenging start*)
	bScavFanOp : BOOL; (*scavenging fan operating*)
	xTON_EGScav: TON;						(* Timer Exhaust Gas Scavenging *)
	xTON_EngRun : TON;						(* Timer Engine Running *)
	bTON_EngRun : BOOL;						(* Trigger Engine Running *)
	xR_TRIG_StorePreEGScavValue : R_TRIG;
	xR_TRIG_StoreAftEGScavValue : R_TRIG;
	rT_bScavValve_PreEGScavValue : REAL;	(* Stored air temperature - Pre Exhaust Gas Scavenging  *)
	rT_bScavValve_AftEGScavValue : REAL;	(* Stored air temperature - After Exhaust Gas Scavenging   *)
	bFS_ScavTime : BOOL;
	xTON_AutStartPrep : TON;
	xTON_CloScavVa : TON;
END_VAR
```

### Program Logical/Exhaust/EG_VaCo (IEC, version 4.04.0) - exhaust gas valve control

#### EG_VaCoCyclic.st
```iecst
(*******************************************************************************
EG_VaCo			 exhaust gas valve control

This code is confidential and proprietary to the INNIO Company.
It may not be used in any form, or reproduced in any manner,
without the express written permission of the INNIO Company.
Copyright, INNIO Company, 2019

Customized modifications: -
------------------------

History:
-------
V0.1	03.07.1998	Pa			erstellt
		24.11.1998	Pa			korrekturlesung
V180	29.01.2003	LH			erweitert für ROTORK-Klappen
V2073	04.04.2006	LH			Abgasklappensteuerung erweitert für Bypass-/Kesselklappen-Kombination
V220	19.02.2007	LH			ROTORK --> EINS
V2600	06.08.2009	lettenb.	task activation added; task: pb2_reg included
V3.99.0	20.03.2013	lettenb.	pb2 --> EG_VaCo renamed
V4.00.1	10.04.2014				xTON_Valves_24h: NCC T91 added(gruber robert: Kombiklappe und Rückmeldung für Bypassklappe und Kesselklappe: nach 24h bleiben die Klappen ständig auf)
		23.06.2014				Para.bSel_EGVa_Combi: overwrite IN_EX.tEG_BoVaOpened.Di/IN_EX.tEG_ByVaOpened.Di removed, bugfix
V4.00.2	12.11.2014				bB_BK_ZU_2C: IN_EX.tEG_BoVaClosedTo.Di -> IN_EX.tEG_ByVaClosedTo.Di, bugfix
								OUT_EX.bEG_ByVaOpened, OUT_EX.bEG_BoVaOpened added, for rel.eng.oper.in heat-regulat. mode
 		07.08.2015  Denk		Manual operating auxiliaries control functionality added
V4.04.0	05.07.2016	lettenb.	xTON_CmdBypassValve_Open.PT: 60s -> 0,5s, bugfix
        20.09.2016				AF_KKAUF: VIS2MM interfaces added for plan(BOP)pictures(mayer robert)
        02.08.2017	lettenb.	INIT added, AF_KKAUF logic changed(validation mayer robert)bu03

Instructions FOR use:
--------------------
Outstandings:
------------
*******************************************************************************)
PROGRAM _INIT
	VIS2MM.bEGValve_Remote := TRUE;
END_PROGRAM

PROGRAM _CYCLIC

	(* Rung 2 *)
	IF Para.bEGValveEnable THEN
		(* Rung 3 *)
		(*----------------------------------------------------------------------------------------*)
		IF NOT Para.bEGValveRegulation THEN  (* exhaust gas valves open/close control *)

			(* DREH_MOM := TRUE AND NOT ROTORK; *)
			DREH_MOM := NOT Para.bSel_EGVa_ROTORK;

			IF Para.bSel_EGVa_Combi THEN (* only bypass valve feedback signales *)
				BYPASS := IN_EX.tEG_ByVaOpened.Di;(* Position Bypass *)
				KESSEL := IN_EX.tEG_ByVaClosed.Di;(* Position Boiler *)
			ELSE
				BYPASS := IN_EX.tEG_BoVaClosed.Di;(* Position Bypass *)
				KESSEL := IN_EX.tEG_ByVaClosed.Di;(* Position Boiler *)
			END_IF;

			(* Demand Boiler valve open *)
			AF_KKAUF := IN_EX.tEng_Run.Do
				AND   ((NOT IN_EX.tEG_BypassDemand.Di AND     VIS2MM.bEGValve_Remote)
					OR (NOT VIS2MM.bBypassDemand      AND NOT VIS2MM.bEGValve_Remote));

			(* Control signal Bypass valve AUF *)
			bB_BKAUF_1 := NOT M_KLST_Exh AND NOT B_BKZU AND NOT B_KKAUF;
			bB_BKAUF_2 :=(NOT IN_EX.tEG_ByVaOpened.Di AND NOT Para.bSel_EGVa_Combi) OR (NOT BYPASS AND Para.bSel_EGVa_Combi);
			bB_BKAUF_3 := bB_BKAUF_2 AND (NOT AF_KKAUF  OR T91);
			B_BKAUF    := bB_BKAUF_1 AND bB_BKAUF_3;

			(* Control signal Bypass Valve Close *)
			bB_BK_ZU_1  := NOT M_KLST_Exh AND NOT B_BKAUF AND NOT B_KKZU;
			bB_BK_ZU_2A := NOT IN_EX.tEG_ByVaClosed.Di AND NOT Para.bSel_EGVa_Combi;
			bB_BK_ZU_2B := NOT KESSEL AND Para.bSel_EGVa_Combi;
			bB_BK_ZU_2C := IN_EX.tEG_ByVaClosedTo.Di AND DREH_MOM;
			bB_BK_ZU_2  := bB_BK_ZU_2A OR bB_BK_ZU_2B OR bB_BK_ZU_2C;
			bB_BK_ZU_3  := AF_KKAUF AND NOT T91 AND (IN_EX.tEG_BoVaOpened.Di OR Para.bSel_EGVa_Combi);
			B_BKZU      := bB_BK_ZU_1 AND bB_BK_ZU_2 AND bB_BK_ZU_3;

			(* Control Signal Boiler valve open *)
			bB_KKAUF_1 := NOT M_KLST_Exh AND NOT B_KKZU AND NOT B_BKAUF;
			bB_KKAUF_2 :=(NOT IN_EX.tEG_BoVaOpened.Di AND NOT Para.bSel_EGVa_Combi) OR (NOT KESSEL AND Para.bSel_EGVa_Combi);
			bB_KKAUF_3 := AF_KKAUF OR T91;
			B_KKAUF    := bB_KKAUF_1 AND bB_KKAUF_2 AND bB_KKAUF_3;

			(* Control signal Boiler valve Close *)
			bB_KKZU_1  := NOT M_KLST_Exh AND NOT B_KKAUF AND NOT B_BKZU;
			bB_KKZU_2A := NOT IN_EX.tEG_BoVaClosed.Di AND NOT Para.bSel_EGVa_Combi;
			bB_KKZU_2B := NOT BYPASS AND Para.bSel_EGVa_Combi;
			bB_KKZU_2C := IN_EX.tEG_BoVaClosedTo.Di AND DREH_MOM;
			bB_KKZU_2  := bB_KKZU_2A OR bB_KKZU_2B OR bB_KKZU_2C;
			bB_KKZU_3  := NOT AF_KKAUF AND NOT T91 AND (IN_EX.tEG_ByVaOpened.Di OR Para.bSel_EGVa_Combi);
			B_KKZU     := bB_KKZU_1 AND bB_KKZU_2 AND bB_KKZU_3;

			(* open valves after 24 hours  *)
			IF Para.bSel_EGVa_Combi THEN bZM_1 := KESSEL OR BYPASS;
			ELSE                         bZM_1 := IN_EX.tEG_BoVaClosed.Di OR IN_EX.tEG_ByVaClosed.Di;
			END_IF;
			xTON_Valves_24h(IN:= bZM_1 AND NOT T91, PT:= T#24h);
			xTOF_Valve_5s(IN:= xTON_Valves_24h.Q, PT:= T#5s);	(* open for 5 seconds *)
			T91		:= xTOF_Valve_5s.Q;

			(* Command Open Boiler valve *)
			xTON_BoilerValve_Open(IN:= B_KKAUF AND NOT OUT_EX.tEG_BoVaCoClose.Do, PT:= T#0.5s);
			OUT_EX.tEG_BoVaCoOpen.Do := xTON_BoilerValve_Open.Q
										OR IN_EX.tManAuxCtr.bEG_BoVaCoOpen;		(* Manual operating auxiliaries control - Handbedienebene *)

			(* Command Boiler Timer Values for Open/Close *)
			IF (Para.bSel_EGVa_ROTORK) THEN
				xTOF_BoilerValve_Close.PT    := T#2s; (* Boiler Valve *)
				xTOF_CmdBypassValve_Close.PT := T#2s; (* Bypass Valve *)
			ELSE
				xTOF_BoilerValve_Close.PT    := T#0s;  (* Boiler Valve *)
				xTOF_CmdBypassValve_Close.PT := T#0s;  (* Bypass Valve *)
			END_IF;

			(* Command Boiler valve Close *)
			xTON_BoilerValve_Close(IN:= B_KKZU, PT:= T#0.5s);
			xTOF_BoilerValve_Close.IN := xTON_BoilerValve_Close.Q;
			IF M_KLST_Exh OR B_KKAUF THEN
				xTOF_BoilerValve_Close(IN := FALSE, PT := T#0s);
			ELSE
				xTOF_BoilerValve_Close();
			END_IF;
			OUT_EX.tEG_BoVaCoClose.Do :=   xTOF_BoilerValve_Close.Q
										OR IN_EX.tManAuxCtr.bEG_BoVaCoClose;	(* Manual operating auxiliaries control - Handbedienebene *)

			(* Command Bypass valve open *)
			xTON_CmdBypassValve_Open(IN:= B_BKAUF AND NOT OUT_EX.tEG_ByVaCoClose.Do, PT:= T#0.5s);
			OUT_EX.tEG_ByVaCoOpen.Do :=    xTON_CmdBypassValve_Open.Q
										OR IN_EX.tManAuxCtr.bEG_ByVaCoOpen;		(* Manual operating auxiliaries control - Handbedienebene *)

			(* Command Bypass valve Close *)
			xTON_CmdBypassValve_Close(IN:= B_BKZU, PT:= T#0.5s);
			xTOF_CmdBypassValve_Close.IN := xTON_CmdBypassValve_Close.Q;
			IF M_KLST_Exh AND B_BKAUF THEN
				xTOF_CmdBypassValve_Close(IN := FALSE, PT := T#0s);
			ELSE
				xTOF_CmdBypassValve_Close();
			END_IF;
			OUT_EX.tEG_ByVaCoClose.Do :=   xTOF_CmdBypassValve_Close.Q
										OR IN_EX.tManAuxCtr.bEG_ByVaCoClose;	(* Manual operating auxiliaries control - Handbedienebene *)

			(* Overwrite Notification/Command with Bypass/boiler valve combination *)
			(* Rung 26 *)

		    IF Para.bSel_EGVa_Combi THEN
				(* Overwrite Open Notification Boiler valve *)
	//			IN_EX.tEG_BoVaOpened.Di   := NOT BYPASS;

				(* Overwrite Open Notification Bypass valve *)
	//			IN_EX.tEG_ByVaOpened.Di   := NOT KESSEL;

				(* Overwrite Command for Boiler Operation *)
				AF_KESSEL                 := OUT_EX.tEG_BoVaCoOpen.Do OR OUT_EX.tEG_ByVaCoClose.Do;
				OUT_EX.tEG_BoVaCoOpen.Do  := AF_KESSEL;
				OUT_EX.tEG_ByVaCoClose.Do := AF_KESSEL;

				(* Overwrite command for Bypass Operation *)
				AF_BYPASS                 := OUT_EX.tEG_BoVaCoClose.Do OR OUT_EX.tEG_ByVaCoOpen.Do;
				OUT_EX.tEG_BoVaCoClose.Do := AF_BYPASS;
				OUT_EX.tEG_ByVaCoOpen.Do  := AF_BYPASS;

				OUT_EX.bEG_ByVaOpened := NOT KESSEL;
				OUT_EX.bEG_BoVaOpened := NOT BYPASS;
			ELSE
				OUT_EX.bEG_ByVaOpened := IN_EX.tEG_ByVaOpened.Di;
				OUT_EX.bEG_BoVaOpened := IN_EX.tEG_BoVaOpened.Di;
			END_IF;
		(*----------------------------------------------------------------------------------------*)
		ELSE 	(* exhaust gas valves open/close regulation *)

			(* Request Boiler valve Open *)
			FG_REG := IN_EX.tEng_Run.Do;

			(* Request increase/decrease heat output - interface from MM_CU/plant controller *)
			KL_PLUS  := IN_EX.bEGValCtr_HeatOutputUp;
			KL_MINUS := IN_EX.bEGValCtr_HeatOutputDown;
			// Commented out for test case 16 written directly

			(* Control signal Bypass Valve Open *)
			B_BKAUF_1 := NOT FG_REG OR (IN_EX.tEng_Run.Do AND KL_MINUS);
			B_BKAUF   := NOT M_KLST_Exh AND B_BKAUF_1 AND NOT IN_EX.tEG_ByVaOpened.Di AND NOT B_BKZU;

			(* Control signal Bypass valve Close *)
			bB_BKZU_1 := NOT M_KLST_Exh AND IN_EX.tEng_Run.Do AND KL_PLUS;
			bB_BKZU_2 := IN_EX.tEG_BoVaOpened.Di AND NOT IN_EX.tEG_ByVaClosed.Di AND NOT B_BKAUF;
			B_BKZU    := bB_BKZU_1 AND bB_BKZU_2;

			(* Control signal Boiler valve Open *)
			b_B_KKAUF_1 := NOT M_KLST_Exh AND IN_EX.tEng_Run.Do AND KL_PLUS;
			b_B_KKAUF_2 := NOT IN_EX.tEG_BoVaOpened.Di AND NOT B_KKZU;
			B_KKAUF     := b_B_KKAUF_1 AND b_B_KKAUF_2;

			(* Control signal Boiler valve Close  *)
			b_B_KKZU_1 := IN_EX.tEG_ByVaOpened.Di AND NOT IN_EX.tEG_BoVaOpened.Di AND B_KKAUF;
			b_B_KKZU_2 := NOT FG_REG OR (IN_EX.tEng_Run.Do AND KL_MINUS);
			B_KKZU     := NOT M_KLST_Exh AND b_B_KKZU_1 AND b_B_KKZU_2;

			(* Command Boiler valve Open *)
			OUT_EX.tEG_BoVaCoOpen.Do  := B_KKAUF;

			(* Command Boiler valve Close *)
			OUT_EX.tEG_BoVaCoClose.Do := B_KKZU;

			(* Command Bypass valve Open *)
			OUT_EX.tEG_ByVaCoOpen.Do  := B_BKAUF;

			(* Command Bypass valve Close *)
			OUT_EX.tEG_ByVaCoClose.Do := B_BKZU;

			(* release engine operation from EG valves *)
			OUT_EX.bEG_ByVaOpened := IN_EX.tEG_ByVaOpened.Di;
			OUT_EX.bEG_BoVaOpened := IN_EX.tEG_BoVaOpened.Di;

		END_IF;
	ELSE
		(* release engine operation from EG valves *)
		OUT_EX.bEG_ByVaOpened := TRUE;
		OUT_EX.bEG_BoVaOpened := TRUE;
	END_IF;

END_PROGRAM
```

#### EG_VaCo.var
```iecst
VAR
	b_B_KKAUF_1 : BOOL := FALSE;
	b_B_KKAUF_2 : BOOL := FALSE;
	b_B_KKZU_1 : BOOL := FALSE;
	b_B_KKZU_2 : BOOL := FALSE;
	B_BKAUF_1 : BOOL := FALSE;
	bB_BK_ZU_1 : BOOL := FALSE;
	bB_BK_ZU_2 : BOOL := FALSE;
	bB_BK_ZU_2A : BOOL := FALSE;
	bB_BK_ZU_2B : BOOL := FALSE;
	bB_BK_ZU_2C : BOOL := FALSE;
	bB_BK_ZU_3 : BOOL := FALSE;
	bB_BKAUF_1 : BOOL := FALSE;
	bB_BKAUF_2 : BOOL := FALSE;
	bB_BKAUF_3 : BOOL := FALSE;
	bB_BKZU_1 : BOOL := FALSE;
	bB_BKZU_2 : BOOL := FALSE;
	bB_KKAUF_1 : BOOL := FALSE;
	bB_KKAUF_2 : BOOL := FALSE;
	bB_KKZU_1 : BOOL := FALSE;
	bB_KKZU_2 : BOOL := FALSE;
	bB_KKZU_3 : BOOL := FALSE;
	bZM_1 : BOOL := FALSE;
	xTOF_BoilerValve_Close : TOF := (0);
	xTOF_CmdBypassValve_Close : TOF := (0);
	xTOF_Valve_5s : TOF := (0);
	xTON_BoilerValve_Close : TON := (0);
	xTON_BoilerValve_Open : TON := (0);
	xTON_CmdBypassValve_Close : TON := (0);
	xTON_CmdBypassValve_Open : TON := (0);
	xTON_Valves_24h : TON := (0);
	bB_KKZU_2A : BOOL;
	bB_KKZU_2B : BOOL;
	bB_KKZU_2C : BOOL;
	bB_KKAUF_3 : BOOL;
END_VAR
```

### Program Logical/Exhaust/Pr_EG_TC1 (IEC, version 4.07.0) - fast exhaust gas pressure sensor

#### Pr_EG_TC1Cyclic.st - Zyklischer Code
```iecst
(*******************************************************************************
Pr_EG_TC1	Fast exhaust gas pressure sensor operations

This code is confidential AND proprietary to the INNIO Company.
It may NOT be used in any form, or reproduced in any manner,
without the express written permission of the INNIO Company.
Copyright, INNIO Company, 2019

Customized modifications: -
------------------------

History:
-------
V4.05.0	29.11.2017	Messner		new created
		04.12.2017	Messner		OXicat inlet pressure fast sensor operation added
V4.07.0	14.01.2019	Schmid		exhaust gas pressure fast (deflagration detection) fully replaces OXIcat inlet pressure fast sensor
								TASK RENAMED: New name: Pr_EG_TC1 - Fast exhaust gas pressure sensor operations
										 (Old name: CAT - Oxidation Catalyst sensor operations)
								-> functionality identical, parameters + MM2VIS vars reused, local vars renamed and new IO label
		18.03.2019	lettenb.	IN_EX.bEng_Start -> IN_EX.bEng_Start_TC1, tPr_EG_Deflag_Fast -> tPr_EG_Deflag_Fast_TC1, mapping + taskclass corr.
V4.14.0	16.10.2024	VighM		Deflagration set cleanup and warning update, minimum peak detection added

Instructions FOR use:
--------------------
- Used for fast sensor operations (Cyclic #1 - at least 5ms)

Outstandings:
------------
*******************************************************************************)

PROGRAM _CYCLIC

	(*===========================================================================*)
	(* Exhaust gas pressure fast operation (deflagration detection) *)
	(*===========================================================================*)

	(* Rising Edge on exhaust gas pressure maximum *)
	xR_TRIG_Pr_EG_Deflag_Fast(CLK:= Para.bPr_OXIcat_In_Fast_Exist		(*Parameter from "OXIcat inlet pressure fast" reused*)
								AND IN_EX.tPr_EG_Deflag_Fast_TC1.GoodQual AND NOT MM2VIS.bMsg9249	(*Good signal quality and no signal warning*)
								AND IN_EX.tPr_EG_Deflag_Fast_TC1.Ai >= Para.rPr_EG_Deflag_Fast_HiHi	(*Exceeding pressure limit*)
								AND ((IN_EX.rN_EngAct_TC1 > 0) OR IN_EX.bEng_Start_TC1)				(*Engine demand or engine moving*)
								AND NOT bPr_EG_Deflag_Fast);										(*Deflagration detected based on first pressure limit exceeding*)

	(* set exhaust gas pressure fast maximum trigger *)
	IF 	xR_TRIG_Pr_EG_Deflag_Fast.Q	THEN

		(* set Msg trigger *)
		bPr_EG_Deflag_Fast := TRUE;

	END_IF;

	(*---------------------------------------------------------------------------*)
	(* Exhaust gas pressure fast peak detection *)
	xTOF_Pr_EG_Deflag_Fast(IN := xR_TRIG_Pr_EG_Deflag_Fast.Q, PT := T#200ms);

	(* continous maximum peak detection *)
	IF 		xTOF_Pr_EG_Deflag_Fast.Q
		AND IN_EX.tPr_EG_Deflag_Fast_TC1.Ai > MM2VIS.rPr_OXIcat_In_Fast_Peak THEN

		(* set new peak pressure value *)
		MM2VIS.rPr_OXIcat_In_Fast_Peak := IN_EX.tPr_EG_Deflag_Fast_TC1.Ai;	(*MM2VIS variable from "OXIcat inlet pressure fast" reused*)
	END_IF;

	(*continous minimum detection*)
	IF 		xTOF_Pr_EG_Deflag_Fast.Q
		AND IN_EX.tPr_EG_Deflag_Fast_TC1.Ai < MM2VIS.rPr_OXIcat_In_Fast_Minimum THEN

		(* set new peak pressure value *)
		MM2VIS.rPr_OXIcat_In_Fast_Minimum := IN_EX.tPr_EG_Deflag_Fast_TC1.Ai;
	END_IF;

	(*---------------------------------------------------------------------------*)
	(* reset exhaust gas pressure fast maximum trigger variables - continuous set is prevented in alarm set condition*)
	IF bPr_EG_Deflag_Fast AND EDGENEG(MM2VIS.bMsg2340) THEN
		bPr_EG_Deflag_Fast := FALSE;
	END_IF;

	(* delayed reset of exhaust gas pressure fast maximum MM2VIS variables *)
	(* to ensure registration of peak values on myPlant *)
	xTOF_Pr_EG_Deflag_Fast_VisReset(IN:= EDGENEG(xTOF_Pr_EG_Deflag_Fast.Q), PT:= T#1m);
	IF EDGENEG(xTOF_Pr_EG_Deflag_Fast_VisReset.Q) THEN
		MM2VIS.rPr_OXIcat_In_Fast_Peak	:= 0;		(*MM2VIS variable from "OXIcat inlet pressure fast" reused*)
		MM2VIS.rPr_OXIcat_In_Fast_Minimum	:= Para.rPr_OXIcat_In_Fast_ScalMax;	(*Update minimum monitoring value to deflagration pressure limit*)
	ELSIF NOT (xTOF_Pr_EG_Deflag_Fast.Q) AND NOT (xTOF_Pr_EG_Deflag_Fast_VisReset.Q) THEN
		MM2VIS.rPr_OXIcat_In_Fast_Minimum	:= Para.rPr_OXIcat_In_Fast_ScalMax;	(*Update minimum monitoring value to deflagration pressure limit*)
	END_IF;

END_PROGRAM
```

#### Pr_EG_TC1.var - Lokale Variablen
```iecst
VAR
	xR_TRIG_Pr_EG_Deflag_Fast : R_TRIG;	(* Rising edge - Trigger on exhaust gas pressure fast *) (*OldName:xR_TRIG_Pr_OXIcat_In_Fast; Cycle:1*)
	xTOF_Pr_EG_Deflag_Fast_VisReset : TOF;
END_VAR
```

### Program Logical/Exhaust/codinox (IEC, version 4.03.0) - Codinox

#### codinoxCyclic.st
```iecst
(*******************************************************************************
codinox		codinox control

This code is confidential and proprietary to the INNIO Company.
It may not be used in any form, or reproduced in any manner,
without the express written permission of the INNIO Company.
Copyright, INNIO Company, 2019

Customized modifications: -
------------------------

History:
-------
V0.1	27.06.2001/LH		erstellt
V0.2	14.02.2003/Wa		Drehmomentschalter entfernt, Ausgabe WatchDog,
 							Umschaltung CODINOX, Sammelstörung CO2
V190	29.07.2004/LH		überarbeitet für Modulisierung
V220	19.02.2007/LH		angepasst für X20-Einführung
V220.1	10.07.2007/Wa		-Vorbereitung für pneumatische CO2-Klappe
 							-Variante für Temp. nach WT2 über Pt100
 							-Deaktivierung der Störungen,
 			 				 wenn CODINOX über Parameter deaktiviert wird
 							-Blockierung CO2-Klappe hinzu
 							-Anzeige der Abgastemp in P50 aktivieren,
 			 				 falls kein Codinox vorhanden
V2.20.2	29.08.2008/PN		-Anzeige der Abgastemp in P50 entfernt,
 			 				da Anzeige im Bild P_312
V3.20.0	30.09.2010/MM(BuR)	M_GSEIN durch GCB_ON ersetzt
		30.09.2010/MM(BuR) 	gen_sch durch GCB_ON_TC1 ersetzt
		01.10.2010 MM(BuR) 	net_sch durch MCB_ON ersetzt
		17.12.2010 lettenb.	RESET_COV, RESET_CO2 removed, autoreset in task: alarms35xx
V4.00.0	18.02.2014			start/stop part load operation from new DI(gridcode)
V4.00.1	24.09.2014			tCO2_Alarm.Do,tCO2_Rdy.Do: old var changed, bugfix
V4.03.0	12.11.2015 Denk		Manual operating auxiliaries control - Handbedienebene for BEL/HOL

Instructions for use:
--------------------
Outstandings:
------------
*******************************************************************************)
PROGRAM _CYCLIC

	(* Variation codinox with pneumatic CO2 valve *)
	Para.bCO2_PneumVal;

	(* digital in from gridcode *)
								IN_EX.tP_GenC_SetEUCOn.Di; 		(* DI: request power value from EU - on (activate) *) (* OldName: DI_GCP_P_S; Cycle:HALioDi_Type; *)
								IN_EX.tP_GenC_SetEUCOf.Di; 		(* DI: request power value from EU - off (deactivate) *) (* OldName: DI_GCP_P_R; Cycle:HALioDi_Type; *)
	P_GenC_SetFixEU[1]		:=	IN_EX.tP_GenC_SetFix1EU.Di; 	(* DI: power value - P- fixvalue 1 from EU *) (* OldName: DI_GCP_P_FIX1; Cycle:HALioDi_Type; *)
	P_GenC_SetFixEU[2]		:=	IN_EX.tP_GenC_SetFix2EU.Di; 	(* DI: power value - P- fixvalue 2 from EU *) (* OldName: DI_GCP_P_FIX2; Cycle:HALioDi_Type; *)
	P_GenC_SetFixEU[3]		:=	IN_EX.tP_GenC_SetFix3EU.Di; 	(* DI: power value - P- fixvalue 3 from EU *) (* OldName: DI_GCP_P_FIX3; Cycle:HALioDi_Type; *)
	P_GenC_SetFixEU[4]		:=	IN_EX.tP_GenC_SetFix4EU.Di; 	(* DI: power value - P- fixvalue 4 from EU *) (* OldName: DI_GCP_P_FIX4; Cycle:HALioDi_Type; *)
	P_GenC_SetFixEU[5]		:=	IN_EX.tP_GenC_SetFix5EU.Di; 	(* DI: power value - P- fixvalue 5 from EU *) (* OldName: DI_GCP_P_FIX5; Cycle:HALioDi_Type; *)
								IN_EX.tPLim_GenC_SetEUCOn.Di; 	(* DI: setpoint power limitation (Plim) from EU - on (activate) *) (* OldName: DI_GCP_Plim_S; Cycle:HALioDi_Type; *)
								IN_EX.tPLim_GenC_SetEUCOf.Di; 	(* DI: setpoint power limitation (Plim) from EU - off (deactivate) *) (* OldName: DI_GCP_Plim_R; Cycle:HALioDi_Type; *)
	PLim_GenC_SetEUPFix[1]	:=	IN_EX.tPLim_GenC_SetEUPFix1.Di;	(* DI: power limitation fixvalue 1 *) (* OldName: DI_EVU_1; Cycle:HALioDi_Type; *)
	PLim_GenC_SetEUPFix[2]	:=	IN_EX.tPLim_GenC_SetEUPFix2.Di;	(* DI: power limitation fixvalue 2 *) (* OldName: DI_EVU_2; Cycle:HALioDi_Type; *)
	PLim_GenC_SetEUPFix[3]	:=	IN_EX.tPLim_GenC_SetEUPFix3.Di;	(* DI: power limitation fixvalue 3 *) (* OldName: DI_EVU_3; Cycle:HALioDi_Type; *)
	PLim_GenC_SetEUPFix[4]	:=	IN_EX.tPLim_GenC_SetEUPFix4.Di;	(* DI: power limitation fixvalue 4 *) (* OldName: DI_EVU_4; Cycle:HALioDi_Type; *)
	PLim_GenC_SetEUPFix[5]	:=	IN_EX.tPLim_GenC_SetEUPFix5.Di;	(* DI: power limitation fixvalue 5 *) (* OldName: DI_EVU_5; Cycle:HALioDi_Type; *)

	(* Codinox available *)
	IF NOT Para.bCodinox_Active THEN

		IN_EX.tT_CO2_Hi.Di        := FALSE;
		CO2KLST_W 				  := FALSE;
		CO2KLST_A 				  := FALSE;
		IN_EX.tCO2_FanFailure.Di  := FALSE;
		IN_EX.tCO2_DevFailure.Di  := FALSE;

		OUT_EX.tCO2_Rdy.Do        := FALSE;

	ELSE
	    (* Notification CO2_Exh flap closed  *)
	    M_KZU := IN_EX.tCO2_VaClosed.Di;

	    (* Notification CO2_Exh flap opened  *)
	    M_KAUF := IN_EX.tCO2_VaOpened.Di;

	    (* Release for CO2_Exh *)
	    FG_CO2 := Para.bCodinox_Active AND IN_EX.tGCB_On.Di AND NOT bGnlTrip AND NOT MM2VIS.bMsg3511;

		(* start/end part load operation *)
		bStartPartLoad := FALSE;
		bStopPartLoad  := FALSE;

		FOR x:=1 TO 5 DO
			xR_TRIG_P_GenC_SetFixEU[x](CLK:= P_GenC_SetFixEU[x]);
			xF_TRIG_P_GenC_SetFixEU[x](CLK:= P_GenC_SetFixEU[x]);
			xR_TRIG_PLim_GenC_SetEUPFix[x](CLK:= PLim_GenC_SetEUPFix[x]);
			xF_TRIG_PLim_GenC_SetEUPFix[x](CLK:= PLim_GenC_SetEUPFix[x]);

			IF xR_TRIG_P_GenC_SetFixEU[x].Q OR xR_TRIG_PLim_GenC_SetEUPFix[x].Q THEN bStartPartLoad := TRUE;
			END_IF;
			IF xF_TRIG_P_GenC_SetFixEU[x].Q OR xF_TRIG_PLim_GenC_SetEUPFix[x].Q THEN bStopPartLoad := TRUE;
			END_IF;
		END_FOR;

		(* interrupt demand codinox at start part load operation for xx sec *)
	    xTP_TEILLAST_START(IN:= bStartPartLoad, PT:= Para.tiCO2_ExPSp_StartOffTime);
		TEILLAST_START := xTP_TEILLAST_START.Q AND AUTO AND AWS_F;

	    (* interrupt demand codinox at end part load operation for xx sec *)
	    xTP_TEILLAST_ENDE(IN:= bStopPartLoad, PT:= Para.tiCO2_ExPSp_StopOffTime);
		TEILLAST_ENDE := xTP_TEILLAST_ENDE.Q AND AUTO AND AWS_F;

	    (* Demand CO2_Exh *)
	    xTON_AFCO2(IN:= FG_CO2 AND IN_EX.tCO2_Demand.Di AND NOT TEILLAST_START AND NOT TEILLAST_ENDE, PT:= T#5s);
		AF_CO2 := xTON_AFCO2.Q;

	    (* Demand CODINOX *)
	    xRS_ANF_CODI.SET := xTON_AFCO2.Q;
		xRS_ANF_CODI.RESET1 := NOT AF_CO2 AND (M_KZU OR MM2VIS.bMsg3314);
		xRS_ANF_CODI();
	    OUT_EX.tCO2_DemCodinox.Do := xRS_ANF_CODI.Q1
									 OR IN_EX.tManAuxCtr.bCO2_DemCodinox;	(* Manual operating auxiliaries control - Handbedienebene *)

	    (* Demand CO2_Exh flap advance open *)
	    xTOF_AFKAUF(IN:= AF_CO2 AND IN_EX.tCodinox_Rdy.Di AND NOT IN_EX.tCO2_VaLockout.Di, PT:= T#1s);
		AF_KAUF := xTOF_AFKAUF.Q;

	    (* command CO2_Exh flap open *)
		B_KAUF := 	Para.bCodinox_Active
			AND NOT MM2VIS.bMsg3314
			AND NOT MM2VIS.bMsg3512
			AND 	AF_KAUF
			AND NOT B_KZU
			AND(NOT M_KAUF OR Para.bCO2_PneumVal);

	    (* command CO2 flap close *)
		B_KZU :=	Para.bCodinox_Active
			AND NOT MM2VIS.bMsg3314
			AND NOT AF_KAUF
			AND NOT B_KAUF
			AND NOT M_KZU;

	    (* Command CO2 flap open *)
		xTON_CO2KAUF(IN := B_KAUF, PT := T#0.5s);
		OUT_EX.tCO2_VaCoOpen.Do := xTON_CO2KAUF.Q;

	    (* Command CO2 flap close *)
	    xTON_CO2KZU(IN:= B_KZU, PT:= T#0.5s);
		OUT_EX.tCO2_VaCoClose.Do := xTON_CO2KZU.Q;

	    (* CO2 Fan ON *)
	    OUT_EX.tCO2_FanCoOn.Do := AF_KAUF AND M_KAUF AND NOT MM2VIS.bMsg3510;

	    (* CO2 Flap disturbance *)
	    xTON_KLST_a(IN:= NOT M_KZU AND OUT_EX.tCO2_VaCoClose.Do, PT:= T#35s);
		ZM_KLSTA := xTON_KLST_a.Q;

	    xTON_KLST_b(IN := NOT IN_EX.tCO2_VaFailure.Di, PT:= T#2s);
		HM_KLST  := xTON_KLST_b.Q;

	    (* CO2 Flap disturbance with Flap-Close command stoppage *)
	    CO2KLST_A := ZM_KLSTA OR (HM_KLST AND M_KAUF);

	    (* Flap disturbance stoppage *)
		xTON_KLST(IN:= NOT M_KAUF AND OUT_EX.tCO2_VaCoOpen.Do, PT:= T#35s);
		CO2KLST_W := xTON_KLST.Q OR (HM_KLST AND NOT M_KAUF);

	    (* Warning flap disturbance *)
	    OUT_EX.tCO2_MPMode.Do := Para.bCodinox_Active AND IN_EX.tGCB_On.Di AND IN_EX.tMCB_On.Di;

	    (* WatchDog *)
	    OUT_EX.tCO2_WD.Do := IN_EX.tCodinox_Rdy.Di;

	    (*Störung CO2_Exh*)
	    OUT_EX.tCO2_Alarm.Do := MM2VIS.bMsg3313 OR MM2VIS.bMsg3314 OR MM2VIS.bMsg3510 OR MM2VIS.bMsg3511 OR MM2VIS.bMsg3512;
	    OUT_EX.tCO2_Rdy.Do   := NOT OUT_EX.tCO2_Alarm.Do;
	    CODINOX := TRUE;

	END_IF;

	(* out interfaces *)
	OUT_EX.rT_EGaHE1 := IN_EX.tT_EGaHE1.Ai;
	OUT_EX.rT_EGaHE2 := IN_EX.tT_EGaHE2.Ai;

END_PROGRAM
```

#### codinox.var
```iecst
VAR
	xTON_KLST_b : TON := (0);
	xTON_KLST_a : TON := (0);
	xTON_CO2KZU : TON := (0);
	xTON_CO2KAUF : TON := (0);
	xTON_KLST : TON := (0);
	xTOF_AFKAUF : TOF := (0);
	xRS_ANF_CODI : RS := (0);
	xTON_AFCO2 : TON := (0);
	xTP_TEILLAST_ENDE : TP := (0);
	xTP_TEILLAST_START : TP := (0);
	HM_KLST : BOOL := 0; (* HM *)
	ZM_KLSTA : BOOL := 0; (* ZM *)
	TEILLAST_START : BOOL := 0; (*Start Teillastbetrieb*)
	TEILLAST_ENDE : BOOL := 0; (*Ende Teillastbetrieb*)
	P_GenC_SetFixEU : ARRAY[0..5] OF BOOL;
	PLim_GenC_SetEUPFix : ARRAY[0..5] OF BOOL;
	xR_TRIG_P_GenC_SetFixEU : ARRAY[0..5] OF R_TRIG;
	xF_TRIG_P_GenC_SetFixEU : ARRAY[0..5] OF R_TRIG;
	xR_TRIG_PLim_GenC_SetEUPFix : ARRAY[0..5] OF R_TRIG;
	xF_TRIG_PLim_GenC_SetEUPFix : ARRAY[0..5] OF R_TRIG;
	bStartPartLoad : BOOL;
	bStopPartLoad : BOOL;
	x : INT;
END_VAR
```

### Program Logical/Exhaust/MsgEX (IEC, version 4.25.0) - messages
